(****************************************************************************************)
(*							Beckhoff Automation Poland									*)
(*							L_TBConvDwordToBits v1.0									*)
(*									29.02.2007											*)
(* This FB returns the 32 corresponding bit values for an input value of type ”double word” *)
(*_______________________________________________________________________________________*)
FUNCTION_BLOCK L_TBConvDwordToBits
VAR_INPUT
	dwInput: DWORD;
END_VAR
VAR_OUTPUT
	bBit0: BOOL;
	bBit1: BOOL;
	bBit2: BOOL;
	bBit3: BOOL;
	bBit4: BOOL;
	bBit5: BOOL;
	bBit6: BOOL;
	bBit7: BOOL;
	bBit8: BOOL;
	bBit9: BOOL;
	bBit10: BOOL;
	bBit11: BOOL;
	bBit12: BOOL;
	bBit13: BOOL;
	bBit14: BOOL;
	bBit15: BOOL;
	bBit16: BOOL;
	bBit17: BOOL;
	bBit18: BOOL;
	bBit19: BOOL;
	bBit20: BOOL;
	bBit21: BOOL;
	bBit22: BOOL;
	bBit23: BOOL;
	bBit24: BOOL;
	bBit25: BOOL;
	bBit26: BOOL;
	bBit27: BOOL;
	bBit28: BOOL;
	bBit29: BOOL;
	bBit30: BOOL;
	bBit31: BOOL;
END_VAR
VAR
END_VAR

bBit0:=dwInput.0;
bBit1:=dwInput.1;
bBit2:=dwInput.2;
bBit3:=dwInput.3;
bBit4:=dwInput.4;
bBit5:=dwInput.5;
bBit6:=dwInput.6;
bBit7:=dwInput.7;
bBit8:=dwInput.8;
bBit9:=dwInput.9;
bBit10:=dwInput.10;
bBit11:=dwInput.11;
bBit12:=dwInput.12;
bBit13:=dwInput.13;
bBit14:=dwInput.14;
bBit15:=dwInput.15;
bBit16:=dwInput.16;
bBit17:=dwInput.17;
bBit18:=dwInput.18;
bBit19:=dwInput.19;
bBit20:=dwInput.20;
bBit21:=dwInput.21;
bBit22:=dwInput.22;
bBit23:=dwInput.23;
bBit24:=dwInput.24;
bBit25:=dwInput.25;
bBit26:=dwInput.26;
bBit27:=dwInput.27;
bBit28:=dwInput.28;
bBit29:=dwInput.29;
bBit30:=dwInput.30;
bBit31:=dwInput.31;

END_FUNCTION_BLOCK

(* stored: Version 1.1.0.1, ProductVersion 3.1.4026.13, FileIdentifier 7917f6b395d92282d26451e26db1f766c6af1862, FileSignature 1278ed314dae3762a729911deb2b29c6f17ef24ed530f26dcd357190755600f1572e5de76c56a80f7723e69912a8e8cd2d2ebdc95fbaca9c10d41f72a85a023620e1629a56ae8c0e7a3148fa17df54f45eed1092574071f29f6f77b7cdb52c8f8ce5357ae5c7ded4004ebb81238121fde78375079a85b05e7a0e8f8e57b5e9b2b35ad36a0c5b6fea901783184d614bf1d586ed312f887b230becc44b4e49894e0982f78cc146d59eb8c62ed0f74c3b252fb937a2b5881aa967a6c3c9fe09bc9d2284051b495b461f25c3c8ee4a9c25f1348e3c81c38497a9e7d3f719b0e97d271cbdf030787365f88da23beaaf58aebd094987b56bbb01b7cab695dc0631bfe3
   POU L_TBConvDwordToBits: Id {b2641e14-5170-42b8-baa0-20408d75d377}, SpecialFunc None *)
